TYPE ST_GenGridController_get :
STRUCT
	b_active			: BOOL;
	b_faultActive		: BOOL;
	b_gensetHot			: BOOL;
	b_gensetStarting	: BOOL;
	b_ModeTransActive	: BOOL;
	b_ModeTransInhibit	: BOOL;
	b_ModeChanged		: BOOL;
	b_ShowModeTrans		: BOOL;
	b_extGensetMode 	: BOOL;
	b_gensetcontrol		: BOOL;
	e_BreakerMode		: eBreakerOperationMode;
	e_PowerControlMode	: ePowerControlMode;
	e_GensetMode		: eGensetMode;
	e_GensetStartStop	: eGensetStartStop;
	e_state				: eGenGridState;
	e_RunCondition		: eRunCondition;
	events				: ST_GengridController_events;
	
END_STRUCT
END_TYPE

(* stored: Version 1.1.0.1, ProductVersion 3.1.4026.18
   DUT ST_GenGridController_get: Id {5457115d-123e-4aca-b8a3-5feedc04b8b1} *)
